// TIA Portal V20 export
DATA_BLOCK "DB_LoaderFixture"   // DB106
// stored: InstanceOfName FB_LoaderFixture, InstanceOfType FB
"FB_LoaderFixture"
   // VAR_INPUT
   //    iAxisV_Moving : Bool;
   //    iAxisV_InPos : Bool;
   //    iAxisW_Moving : Bool;
   //    iAxisW_InPos : Bool;
   // END_VAR
   // VAR_OUTPUT
   //    oFixtureOpenReq : Bool;
   //    oFixtureCloseReq : Bool;
   //    oLoadGripperOpenReq : Bool;
   //    oUnloadGripperCloseReq : Bool;
   //    oBlowingReq : Bool;
   //    oAxisV_StartReq : Bool;
   //    oAxisV_PosSetPoint : Real;
   //    oAxisW_StartReq : Bool;
   //    oAxisW_PosSetPoint : Real;
   // END_VAR
   // VAR
   //    sFixtureMain : "FB_FixtureUnloadLoad";
   //    sFixtureUnloading { S7_SetPoint := 'True'} : "FB_FixtureUnloading";
   //    sFixtureLoading { S7_SetPoint := 'True'} : "FB_FixtureLoading";
   //    sFixtureBlowing { S7_SetPoint := 'True'} : "FB_FixtureBlowing";
   //    sFixtureRelease { S7_SetPoint := 'True'} : "FB_FixtureRelease";
   //    sFixtureV_Init { S7_SetPoint := 'True'} : "FB_FixtureV_Init";
   //    sFixtureW_Init { S7_SetPoint := 'True'} : "FB_FixtureW_Init";
   //    sAxisVSafePos { S7_SetPoint := 'True'} : LReal;
   //    sStepPauseSeq { S7_SetPoint := 'True'} : Bool;
   // END_VAR
BEGIN
END_DATA_BLOCK
